FUNCTION "FC_SAV" : Void
{ S7_Optimized_Access := 'TRUE' }
VERSION : 0.1
   VAR_INPUT
      Index_Cell : USInt;
      Vitesse : USInt;
   END_VAR

   VAR_IN_OUT
      SurvDosBenne : "S_DOSBENNE";
   END_VAR


BEGIN
	#SurvDosBenne.Dos_Commun.Module_Commun._PtCel._TabCel[#Index_Cell]._SAV := #Vitesse;
END_FUNCTION

